// TIA Portal V16 export
// export: Created 2024-03-28T09:54:29.8998736Z, ExportSetting WithDefaults, DisplayName Totally Integrated Automation Portal, DisplayVersion V16, DisplayName TIA Portal Version Control Interface, DisplayVersion V16, DisplayName TIA Portal Openness, DisplayVersion V16, DisplayName STEP 7 Professional, DisplayVersion V16, DisplayName STEP 7 Safety, DisplayVersion V16, DisplayName WinCC Advanced, DisplayVersion V16
TYPE "UR__O2T_floats"
// stored: IsFailsafeCompliant false
   STRUCT
      Register : Array[0..11] of Real;
   END_STRUCT;
END_TYPE
